{attribute 'qualified_only'}
{attribute 'to_string'}
TYPE E_DATA_STATE :
(
	NULL,
  NO_EXIST,
  INIT        := 10,
  READ        := 20,
  WRITE       := 30
)UINT;
END_TYPE

(* stored: Version 1.1.0.1, ProductVersion 3.1.4026.20
   DUT E_DATA_STATE: Id {b63aa10f-1c01-4042-a13d-f14bdfc6344a} *)
